TYPE ST_Nanotec_HMI EXTENDS ST_HmiFunction :
	STRUCT
		JogFwd	   : Button;
		JogBwd	   : Button;
		Ready	   : BOOL;
		Faulted	   : BOOL;
		ActVelIncr : INT;
	END_STRUCT
END_TYPE

(* stored: Version 1.1.0.1
   DUT ST_Nanotec_HMI: Id {4383fe85-5e5c-4595-b313-f8d5bde2f215} *)
